SYSTEM TEST_SWING (* Test of Swing components *)
  (* Standard: 61499-1 *)
  (* Version 0.0, 2004-06-18, JHC, Rockwell Automation *)
  APPLICATION APP1
  END_APPLICATION
  DEVICE DEV1 : FRAME_DEVICE
    RESOURCE RES1 : PANEL_RESOURCE
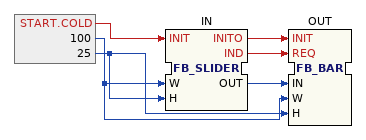
      FBS
        IN : FB_SLIDER;
        OUT : FB_BAR;
      END_FBS
      EVENT_CONNECTIONS
        START.COLD TO IN.INIT;
        IN.INITO TO OUT.INIT;
        IN.IND TO OUT.REQ;
      END_CONNECTIONS
      DATA_CONNECTIONS
        IN.OUT TO OUT.IN;
        100 TO OUT.W;
        25 TO OUT.H;
        100 TO IN.W;
        25 TO IN.H;
      END_CONNECTIONS
    END_RESOURCE
    RESOURCE RES2 : PANEL_RESOURCE
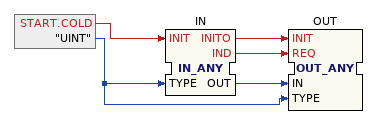
      FBS
        IN : IN_ANY;
        OUT : OUT_ANY;
      END_FBS
      EVENT_CONNECTIONS
        START.COLD TO IN.INIT;
        IN.INITO TO OUT.INIT;
        IN.IND TO OUT.REQ;
      END_CONNECTIONS
      DATA_CONNECTIONS
        IN.OUT TO OUT.IN;
        "UINT" TO IN.TYPE;
        "UINT" TO OUT.TYPE;
      END_CONNECTIONS
    END_RESOURCE
    RESOURCE RES3 : PANEL_RESOURCE
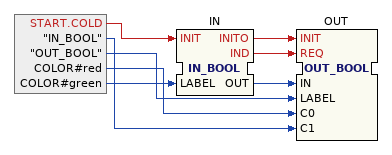
      FBS
        IN : IN_BOOL;
        OUT : OUT_BOOL;
      END_FBS
      EVENT_CONNECTIONS
        START.COLD TO IN.INIT;
        IN.INITO TO OUT.INIT;
        IN.IND TO OUT.REQ;
      END_CONNECTIONS
      DATA_CONNECTIONS
        IN.OUT TO OUT.IN;
        "IN_BOOL" TO IN.LABEL;
        "OUT_BOOL" TO OUT.LABEL;
        COLOR#red TO OUT.C0;
        COLOR#green TO OUT.C1;
      END_CONNECTIONS
    END_RESOURCE
    RESOURCE RES4 : PANEL_RESOURCE
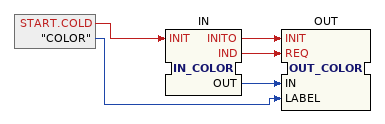
      FBS
        IN : IN_COLOR;
        OUT : OUT_COLOR;
      END_FBS
      EVENT_CONNECTIONS
        START.COLD TO IN.INIT;
        IN.INITO TO OUT.INIT;
        IN.IND TO OUT.REQ;
      END_CONNECTIONS
      DATA_CONNECTIONS
        IN.OUT TO OUT.IN;
        "COLOR" TO OUT.LABEL;
      END_CONNECTIONS
    END_RESOURCE
    RESOURCE RES5 : PANEL_RESOURCE
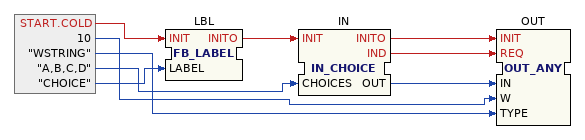
      FBS
        IN : IN_CHOICE;
        OUT : OUT_ANY;
        LBL : FB_LABEL;
      END_FBS
      EVENT_CONNECTIONS
        IN.INITO TO OUT.INIT;
        IN.IND TO OUT.REQ;
        START.COLD TO LBL.INIT;
        LBL.INITO TO IN.INIT;
      END_CONNECTIONS
      DATA_CONNECTIONS
        IN.OUT TO OUT.IN;
        10 TO OUT.W;
        "WSTRING" TO OUT.TYPE;
        "A,B,C,D" TO IN.CHOICES;
        "CHOICE" TO LBL.LABEL;
      END_CONNECTIONS
    END_RESOURCE
    RESOURCE RES6 : PANEL_RESOURCE
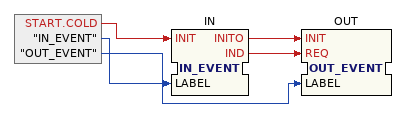
      FBS
        IN : IN_EVENT;
        OUT : OUT_EVENT;
      END_FBS
      EVENT_CONNECTIONS
        START.COLD TO IN.INIT;
        IN.INITO TO OUT.INIT;
        IN.IND TO OUT.REQ;
      END_CONNECTIONS
      DATA_CONNECTIONS
        "IN_EVENT" TO IN.LABEL;
        "OUT_EVENT" TO OUT.LABEL;
      END_CONNECTIONS
    END_RESOURCE
    RESOURCE RES7 : PANEL_RESOURCE
      FBS
        IN : IN_ARRAY;
        OUT : OUT_ARRAY;
      END_FBS
      EVENT_CONNECTIONS
        START.COLD TO IN.INIT;
        IN.INITO TO OUT.INIT;
        IN.IND TO OUT.REQ;
      END_CONNECTIONS
      DATA_CONNECTIONS
        IN.OUT TO OUT.IN;
        5 TO IN.N;
        "UINT" TO IN.TYPE;
        "[1,2,3,4,5]" TO IN.IVAL;
        5 TO OUT.N;
        "UINT" TO OUT.TYPE;
        "[5,4,3]" TO OUT.IVAL;
        10 TO IN.W;
        10 TO OUT.W;
      END_CONNECTIONS
    END_RESOURCE
  END_DEVICE
  DATA_CONNECTIONS (* parameter values *)
    [100,100,250,225] TO DEV1.BOUNDS;
    [7,1] TO DEV1.GRID;
  END_CONNECTIONS
END_SYSTEM
